FUNCTION_BLOCK Forces3
VAR_INPUT
	fOvr			: LREAL;
	Execute 		: BOOL;
END_VAR
VAR_OUTPUT
	AxisReady		: BOOL;
END_VAR
VAR
	fbPower				: MC_Power;
	fbReset 			: MC_Reset;
	PowerAxis1Out		: ST_McOutputs;
	fbMoveVelocity		: MC_MoveVelocity;
	bSensor : BOOL;
	bVelocityExecute	: BOOL;
	rVelocity			: LREAL := 600;
	//userDirection		: MC_Negative_Direction;
	bResetExecute: BOOL;
END_VAR
VAR_IN_OUT

END_VAR

fbPower(
	Axis:= GVL_Conveyer.ConveyerAxis, 
	Enable:= Execute, 
	Enable_Positive:= Execute, 
	Enable_Negative:= Execute, 
	Override:= fOvr, );
	
fbMoveVelocity(
			Axis:= GVL_Conveyer.ConveyerAxis, 
			Execute:= bVelocityExecute,
			Velocity:= rVelocity, 
			Direction := MC_Negative_Direction
			);
fbReset(
		Axis:= GVL_Conveyer.ConveyerAxis,
		Execute := bResetExecute
		);

END_FUNCTION_BLOCK

(* stored: Version 1.1.0.1, ProductVersion 3.1.4024.11
   POU Forces3: Id {1aadb990-287b-47b9-b9e4-71ff077bab8d}, SpecialFunc None *)
